// TIA Portal V20 export
VAR_GLOBAL   // PLC tag table "TROLLEY"
   mhUpperLimitSwitchBypassKeyCh1 AT %I300.0 : Bool;   // MH Upper limit Cam switch bypass key switch Channel 1
   mhUpperLimitSwitchBypassKeyCh2 AT %I300.4 : Bool;   // MH Upper limit Cam switch bypass key switch Channel 2
   mhUpperLimitSwitchBypassKeyCh1VS AT %I301.0 : Bool;   // MH Upper limit Cam switch bypass key switch Channel 1 Supply
   mhUpperLimitSwitchBypassKeyCh2VS AT %I301.4 : Bool;   // MH Upper limit Cam switch bypass key switch Channel 2 Supply
   mhLimitSwitchEmStopCh1 AT %I306.0 : Bool;   // MH Emergency stop limit switch Channel 1
   mh1LimitSwitchFRUEmStop AT %I306.1 : Bool;   // MH1 cam switch Raise emergency stop
   machineRoomDoorControlCh1 AT %I306.2 : Bool;   // Machine room door control switch Channel 1
   mh2LimitSwitchFRUEmStop AT %I306.3 : Bool;   // MH2 cam switch Raise emergency stop
   mhLimitSwitchEmStopCh2 AT %I306.4 : Bool;   // MH Emergency stop limit switch Channel 2
   mh1LimitSwitchBLDEmStop AT %I306.5 : Bool;   // MH1 cam switch Lower emergency stop
   machineRoomDoorControlCh2 AT %I306.6 : Bool;   // Machine room door control switch Channel 2
   mh2LimitSwitchBLDEmStop AT %I306.7 : Bool;   // MH2 cam switch Lower emergency stop
   machineRoomDoorControlCh1VS AT %I307.2 : Bool;   // Machine room door control switch Channel 1 supply
   mhLimitSwitchEmStopCh2VS AT %I307.4 : Bool;   // MH Emergency stop limit switch Channel 2 supply
   machineRoomDoorControlCh2VS AT %I307.6 : Bool;   // Machine room door control switch Channel 2 supply
   slewLimitSwitchBLDStopCh1 AT %I312.2 : Bool;   // Slewing limit switch Stop left Channel 1
   slewLimitSwitchFRUStopCh1 AT %I312.3 : Bool;   // Slewing limit switch Stop right Channel 1
   slewLimitSwitchBLDStopCh2 AT %I312.6 : Bool;   // Slewing limit switch Stop left Channel 2
   slewLimitSwitchFRUStopCh2 AT %I312.7 : Bool;   // Slewing limit switch Stop right Channel 2
   slewLimitSwitchBLDStopVS AT %I313.2 : Bool;   // Slewing limit switch Stop left Sensor supply
   slewLimitSwitchFRUStopVS AT %I313.3 : Bool;   // Slewing limit switch Stop right Sensor supply
   trolleyEntranceGateSouthControlCh1 AT %I318.2 : Bool;   // Trolley entrance gate south side control Channel 1
   trolleyEntranceGateNorthControlCh1 AT %I318.3 : Bool;   // Trolley entrance gate north side control Channel 1
   trolleyEntranceGateSouthControlCh2 AT %I318.6 : Bool;   // Trolley entrance gate south side control Channel 2
   trolleyEntranceGateNorthControlCh2 AT %I318.7 : Bool;   // Trolley entrance gate north side control Channel 2
   trolleyEntranceGateSouthControlCh1VS AT %I319.2 : Bool;   // Trolley entrance gate south side control Channel 1 supply
   trolleyEntranceGateNorthControlCh1VS AT %I319.3 : Bool;   // Trolley entrance gate north side control Channel 1 supply
   trolleyEntranceGateSouthControlCh2VS AT %I319.6 : Bool;   // Trolley entrance gate south side control Channel 2 supply
   trolleyEntranceGateNorthControlCh2VS AT %I319.7 : Bool;   // Trolley entrance gate north side control Channel 2 supply
   btnEmStopRopeChangeBoxCh1 AT %I324.2 : Bool;   // Rope change box Emergency stop Channel 1
   ropeChangeBoxHoldToRunBtnCh1 AT %I324.3 : Bool;   // Rope change box Hold-to-run button Channel 1
   btnEmStopRopeChangeBoxCh2 AT %I324.6 : Bool;   // Rope change box Emergency stop Channel 2
   ropeChangeBoxHoldToRunBtnCh2 AT %I324.7 : Bool;   // Rope change box Hold-to-run button Channel 2
   btnEmStopRopeChangeBoxCh1VS AT %I325.2 : Bool;   // Rope change box Emergency stop Channel 1 Supply
   ropeChangeBoxHoldToRunBtnCh1VS AT %I325.3 : Bool;   // Rope change box Hold-to-run button Channel 1 Supply
   btnEmStopRopeChangeBoxCh2VS AT %I325.6 : Bool;   // Rope change box Emergency stop Channel 2 Supply
   ropeChangeBoxHoldToRunBtnCh2VS AT %I325.7 : Bool;   // Rope change box Hold-to-run button Channel 2 Supply
   cabinPlatformGateTrolleySideControlCh1 AT %I330.1 : Bool;   // Cabin platform gate (trolley side) control Channel 1
   btnEmStopSpreader AT %I330.2 : Bool;   // Spreader Emergency stop
   cabinEntranceInterlockMagnetPosCh1 AT %I330.3 : Bool;   // Cabin entrance interlock magnet position Channel 1
   cabinPlatformGateTrolleySideControlCh2 AT %I330.5 : Bool;   // Cabin platform gate (trolley side) control Channel 2
   limitSwitchSpreaderAntiTwoBlock AT %I330.6 : Bool;   // Spreader anti-two block emergency switch
   cabinEntranceInterlockMagnetPosCh2 AT %I330.7 : Bool;   // Cabin entrance interlock magnet position Channel 2
   cabinPlatformGateTrolleySideControlCh1VS AT %I331.1 : Bool;   // Cabin platform gate (trolley side) control Channel 1 supply
   btnEmStopSpreaderVS AT %I331.2 : Bool;   // Spreader Emergency stop Channel supply
   cabinPlatformGateTrolleySideControlCh2VS AT %I331.5 : Bool;   // Cabin platform gate (trolley side) control Channel 2 supply
   limitSwitchSpreaderAntiTwoBlockVS AT %I331.6 : Bool;   // Spreader anti-two block emergency switch Channel supply
   spare AT %I360.1 : Bool;   // Spare
   cbIllumSocketsTrolley AT %I360.2 : Bool;   // Illumination/sockets trolley CB Feedback
   cb230VCircuitsTrolley AT %I360.3 : Bool;   // 230V circuits trolley CB Feedback
   cbCabin400VLoads AT %I360.4 : Bool;   // Cabin 400V loads CB Feedback
   cbCabin230VLoads AT %I360.5 : Bool;   // Cabin 230V loads CB Feedback
   cbIllumTrolleyRCB AT %I360.6 : Bool;   // Illumination Trolley RCB Feedback
   cbTrolleySockets400VRCBO AT %I360.7 : Bool;   // Trolley Sockets 400V RCBO Feedback
   cbTrolleySockets230VRCBO AT %I361.0 : Bool;   // Trolley Sockets 230V RCBO Feedback
   cbIllumTrolleyMachineRoom AT %I361.1 : Bool;   // Illumination Trolley machine room CB Feedback
   cbIllumTrolleyWalkways AT %I361.2 : Bool;   // Illumination Trolley walkways CB Feedback
   cbIllumTrolleyFloodLight AT %I361.3 : Bool;   // Illumination Trolley flood light CB Feedback
   cbUpsOutput AT %I361.4 : Bool;   // UPS output CB Feedback
   illumTrolleyFloodLightMCStarted AT %I361.5 : Bool;   // Illumination Trolley flood light contactor Feedback
   upsTrolleyFloodAlarm AT %I361.6 : Bool;   // Trolley flood UPS Alarm
   upsTrolleyFloodBatteryMode AT %I361.7 : Bool;   // Trolley flood UPS Battery mode
   cb24trolleyPS AT %I362.0 : Bool;   // 24VDC Trolley PS CB Feedback
   trolleyPS24OK AT %I362.1 : Bool;   // 24VDC Trolley PS OK
   ups24trolleyBatteryMode AT %I362.2 : Bool;   // 24VDC Trolley UPS Battery mode
   ups24trolleyOK AT %I362.3 : Bool;   // 24VDC Trolley UPS 24VDC OK
   ups24trolleyAlarm AT %I362.4 : Bool;   // 24VDC Trolley UPS Alarm
   ups24trolleyReadyToBuffer AT %I362.5 : Bool;   // 24VDC Trolley UPS Ready to buffer
   ups24trolleyBatGt85 AT %I362.6 : Bool;   // 24VDC Trolley UPS BAT.>85%
   "cbPnSwitchSupply(1)" AT %I362.7 : Bool;   // PN switch supply CB Feedback
   cb24Spare AT %I363.0 : Bool;   // 24 VDC CB Spare Feedback
   "cbAccessCircuits(1)" AT %I363.1 : Bool;   // Access circuits CB Feedback
   cbMotorProtectionRelays AT %I363.2 : Bool;   // Motor protection relays, optic transmitters CB Feedback
   cbMhSensorsSupply AT %I363.3 : Bool;   // MH sensors supply CB Feedback
   "cbCtSensorsSupply(1)" AT %I363.4 : Bool;   // CT sensors supply CB Feedback
   cbSlewSensorsSupply AT %I363.5 : Bool;   // Slewing sensors supply CB Feedback
   cbWindTransmitterSupply AT %I363.6 : Bool;   // Wind transmitter supply CB Feedback
   cbTelephoneSystemTrolley AT %I363.7 : Bool;   // Telephone system supply trolley CB Feedback
   cbLehnertSystem AT %I364.0 : Bool;   // LEHNERT system CB Feedback
   cbLaseIPCSupply AT %I364.1 : Bool;   // LASE IPC supply CB Feedback
   cb230Spare AT %I364.2 : Bool;   // 230V spare CB Feedback
   "cb230Spare(1)" AT %I364.3 : Bool;   // 230V spare CB Feedback
   "cb24Spare(1)" AT %I364.4 : Bool;   // 24VDC spare CB Feedback
   "cb24Spare(2)" AT %I364.5 : Bool;   // 24VDC spare CB Feedback
   cbSiren AT %I364.6 : Bool;   // Siren CB Feedback
   trolleyCoolingFanMCStarted AT %I365.4 : Bool;   // Trolley machine room cooling fan contactor Feedback
   trolleyHeaterMCStarted AT %I365.5 : Bool;   // Trolley machine room heater contactor Feedback
   cbCabinCtrlCircuits24VS AT %I365.6 : Bool;   // Cabin control circuits 24VDC Supply CB Feedback
   cbMh1Brake AT %I366.0 : Bool;   // MH1 Brake CB Feedback
   cbMh1ForcedCoolingFan AT %I366.1 : Bool;   // MH1 Forced cooling fan CB Feedback
   cbMh1AntiCondHeating AT %I366.2 : Bool;   // MH1 Anti- condensation heating CB Feedback
   mh1CoolingFanMCStarted AT %I366.3 : Bool;   // MH1 Forced cooling fan contactor Feedback
   "cbMh1AntiCondHeating(1)" AT %I366.4 : Bool;   // MH1 Anti-condensation heating CB Feedback
   mh1BrakeMC1Started AT %I366.5 : Bool;   // MH1 brake contactor 1 feedback
   mh1BrakeMC2Started AT %I366.6 : Bool;   // MH1 brake contactor 2 feedback
   mh1BrakeOpen AT %I366.7 : Bool;   // MH1 Brake Open
   mh1BrakeWear AT %I367.0 : Bool;   // MH1 Brake Wear
   mh1LimitSwitchFRUStop AT %I367.1 : Bool;   // MH1 cam switch Raise end stop
   mh1LimitSwitchFRUSlowDown AT %I367.2 : Bool;   // MH1 cam switch Raise speed reduction
   mh1LimitSwitchBLDStop AT %I367.3 : Bool;   // MH1 cam switch Lower end stop
   mh1LimitSwitchBLDSlowDown AT %I367.4 : Bool;   // MH1 cam switch Lower speed reduction
   ropeDescendRelay1 AT %I367.6 : Bool;   // Rope descend relay 1
   ropeDescendRelay2 AT %I367.7 : Bool;   // Rope descend relay 2
   cbMh2Brake AT %I368.0 : Bool;   // MH2 Brake CB Feedback
   cbMh2ForcedCoolingFan AT %I368.1 : Bool;   // MH2 Forced cooling fan CB Feedback
   cbMh2AntiCondHeating AT %I368.2 : Bool;   // MH2 Anti- condensation heating CB Feedback
   mh2CoolingFanMCStarted AT %I368.3 : Bool;   // MH2 Forced cooling fan contactor Feedback
   "cbMh2AntiCondHeating(1)" AT %I368.4 : Bool;   // MH2 Anti-condensation heating CB Feedback
   mh2BrakeMC1Started AT %I368.5 : Bool;   // MH2 brake contactor 1 feedback
   mh2BrakeMC2Started AT %I368.6 : Bool;   // MH2 brake contactor 2 feedback
   mh2BrakeOpen AT %I368.7 : Bool;   // MH2 Brake Open
   mh2BrakeWear AT %I369.0 : Bool;   // MH2 Brake Wear
   mh2LimitSwitchFRUStop AT %I369.1 : Bool;   // MH2 cam switch Raise end stop
   mh2LimitSwitchFRUSlowDown AT %I369.2 : Bool;   // MH2 cam switch Raise speed reduction
   mh2LimitSwitchBLDStop AT %I369.3 : Bool;   // MH2 cam switch Lower end stop
   mh2LimitSwitchBLDSlowDown AT %I369.4 : Bool;   // MH2 cam switch Lower speed reduction
   "spare(1)" AT %I369.7 : Bool;   // Spare
   cbCtBrakes AT %I370.0 : Bool;   // CT Brakes CB Feedback
   cbCtAntiCondHeating AT %I370.1 : Bool;   // CT Anti-condensation heating CB Feedback
   ctAntiCondHeatingMCStarted AT %I370.2 : Bool;   // CT Anti-condensation heating contactor Feedback
   ct1Motor1TempCtrl AT %I370.5 : Bool;   // CT1 motor 1 temperature control
   ct1Motor2TempCtrl AT %I370.6 : Bool;   // CT1 motor 2 temperature control
   ct2Motor1TempCtrl AT %I370.7 : Bool;   // CT2 motor 1 temperature control
   ct2Motor2TempCtrl AT %I371.0 : Bool;   // CT2 motor 2 temperature control
   "spare(2)" AT %I371.1 : Bool;   // Spare
   "spare(3)" AT %I371.2 : Bool;   // Spare
   "spare(4)" AT %I371.3 : Bool;   // Spare
   "spare(5)" AT %I371.4 : Bool;   // Spare
   "spare(6)" AT %I371.5 : Bool;   // Spare
   "spare(7)" AT %I371.6 : Bool;   // Spare
   "spare(8)" AT %I371.7 : Bool;   // Spare
   cbSlewBrakes AT %I372.0 : Bool;   // Slewing brakes CB Feedback
   cbSlewAntiCondHeating AT %I372.1 : Bool;   // Slewing anti-condensation heating CB Feedback
   slewAntiCondHeatingMCStarted AT %I372.2 : Bool;   // Slewing anti-condensation heating contactor Feedback
   slewBrakesControlMC1Started AT %I372.3 : Bool;   // Slewing brakes control Contactor 1 feedback
   slewBrakesControlMC2Started AT %I372.4 : Bool;   // Slewing brakes control Contactor 2 feedback
   slewMotor1TempCtrl AT %I372.5 : Bool;   // Slewing motor 1 temperature control
   slewMotor2TempCtrl AT %I372.6 : Bool;   // Slewing motor 2 temperature control
   cbKstBoxSupply AT %I373.0 : Bool;   // KST box supply CB Feedback
   loadMomentGt115 AT %I373.1 : Bool;   // Load moment>115%
   loadMomentGt105 AT %I373.2 : Bool;   // Load moment>105%
   loadMomentGt95 AT %I373.3 : Bool;   // Load moment>95%
   loadGt11t AT %I373.4 : Bool;   // Load>11t
   maxUnitLoad AT %I373.5 : Bool;   // Max. unit load
   excenterAbMinusCd AT %I373.6 : Bool;   // Excenter (A+B)-(C+D)
   ropeLoop AT %I373.7 : Bool;   // Rope loop
   cbSpreaderHydraulicPump1 AT %I374.0 : Bool;   // Spreader Hydraulic pump 1 CB Feedback
   cbSpreaderHydraulicPump2 AT %I374.1 : Bool;   // Spreader Hydraulic pump 2 CB Feedback
   cbSpreaderHeating230Vac AT %I374.2 : Bool;   // Spreader Heating power supply 230VAC CB Feedback
   cbSpreaderControl230Vac AT %I374.3 : Bool;   // Spreader Control voltage 230VAC CB Feedback
   cb24SpreaderSupply AT %I374.4 : Bool;   // Spreader 24VDC power supply CB Feedback
   cbSpreaderEmStopRelays AT %I374.5 : Bool;   // Spreader emergency stop relays CB Feedback
   cbLaseCabinet230V AT %I374.6 : Bool;   // LASE cabinet 230V supply CB Feedback
   "cabinEntranceInterlockMagnetPosNO(1)" AT %I375.0 : Bool;   // Cabin entrance interlock magnet position signaling contact (NO)
   lockOpenBtnCabinSide AT %I375.1 : Bool;   // Lock opening button cabin side
   cabinEntranceDoorInterlockMCStarted AT %I375.2 : Bool;   // Cabin entrance door interlock contactor Feedback
   machineRoomDoorControlFb AT %I375.3 : Bool;   // Machine room door control switch Feedback
   cabinPlatformGateTrolleySideControlFb AT %I375.4 : Bool;   // Cabin platform gate (trolley side) control Feedback
   trolleyEntranceGateSouthControlFb AT %I375.5 : Bool;   // Trolley entrance gate south side control Feedback
   trolleyEntranceGateNorthControlFb AT %I375.6 : Bool;   // Trolley entrance gate north side control Feedback
   trolleyExitGateStairsControl AT %I375.7 : Bool;   // Trolley exit to the stairs gate control
   ropeChangeBoxStart AT %I376.0 : Bool;   // Rope change box Start rope change
   ropeChangeBoxSiren AT %I376.1 : Bool;   // Rope change box Siren control
   ropeChangeBoxMhFRU AT %I376.2 : Bool;   // Rope change box MH up
   ropeChangeBoxMhBLD AT %I376.3 : Bool;   // Rope change box MH down
   ropeChangeBoxCtFRU AT %I376.4 : Bool;   // Rope change box CT forward
   ropeChangeBoxCtBLD AT %I376.5 : Bool;   // Rope change box CT backward
   ropeChangeBoxSlewBLD AT %I376.6 : Bool;   // Rope change box Slewing left rotation
   ropeChangeBoxSlewFRU AT %I376.7 : Bool;   // Rope change box Slewing right rotation
   ropeChangeBoxCtParking AT %I377.0 : Bool;   // Rope change box Cross travel to parking position
   cbLubricationStation230V AT %I377.1 : Bool;   // Lubrication station 230V supply CB Feedback
   lubricationEnable AT %I377.2 : Bool;   // Lubrication station enable
   "spare(9)" AT %I377.3 : Bool;   // Spare
   windAlarmWarning AT %I377.6 : Bool;   // Wind Alarm Unit Warning
   "windAlarmWarning(1)" AT %I377.7 : Bool;   // Wind Alarm Unit Warning
   cbJackScrewMotorNorth AT %I378.0 : Bool;   // Jack-screw motor North side CB Feedback
   jackScrewNorthMCFRUStarted AT %I378.1 : Bool;   // Jack-screw motor North side contactor up Feedback
   jackScrewNorthMCBLDStarted AT %I378.2 : Bool;   // Jack-screw motor North side contactor down Feedback
   cbJackScrewMotorSouth AT %I378.3 : Bool;   // Jack-screw motor South side CB Feedback
   jackScrewSouthMCFRUStarted AT %I378.4 : Bool;   // Jack-screw motor South side contactor up Feedback
   jackScrewSouthMCBLDStarted AT %I378.5 : Bool;   // Jack-screw motor South side contactor down Feedback
   jackScrewNorthMotorTempCtrl AT %I378.6 : Bool;   // Jack-screw north side motor temperature control
   jackScrewSouthMotorTempCtrl AT %I378.7 : Bool;   // Jack-screw south side motor temperature control
   jackScrewNorthUpperPos AT %I379.0 : Bool;   // Jack-screw North side Upper position
   jackScrewNorthLowerPos AT %I379.1 : Bool;   // Jack-screw North side Lower position
   jackScrewSouthUpperPos AT %I379.2 : Bool;   // Jack-screw South side Upper position
   jackScrewSouthLowerPos AT %I379.3 : Bool;   // Jack-screw South side Lower position
   slewBrakeMC1Start AT %Q341.2 : Bool;   // Slewing brakes control Contactor 1
   slewBrakeMC2Start AT %Q341.3 : Bool;   // Slewing brakes control Contactor 2
   spreaderEmStopRelay AT %Q346.0 : Bool;   // Spreader emergency stop relay
   cabinEntranceDoorInterlockMCStart AT %Q346.1 : Bool;   // Cabin entrance door interlock control
   sirenStart AT %Q360.0 : Bool;   // Siren control relay
   mh1CoolingFanMCStart AT %Q360.1 : Bool;   // MH1 cooling fan Contactor
   mh1AntiCondMCStart AT %Q360.2 : Bool;   // MH1 anti-condensation heating Contactor
   mh2CoolingFanMCStart AT %Q360.3 : Bool;   // MH2 cooling fan Contactor
   mh2AntiCondMCStart AT %Q360.4 : Bool;   // MH2 anti-condensation heating Contactor
   ctAntiCondMCStart AT %Q360.5 : Bool;   // CT Anti-condensation heating control Contactor
   slewAntiCondMCStart AT %Q360.6 : Bool;   // Slewing anti-condensation heating control Contactor
   illumTrolleyWalkwaysMCStart AT %Q361.0 : Bool;   // Illumination Trolley walkways ON/OFF (impulse control)
   illumTrolleyFloodLightMCStart AT %Q361.3 : Bool;   // Illumination Trolley flood light ON/OFF (impulse control)
   lubricationStart AT %Q361.6 : Bool;   // Lubrication station control
   lubricationAddStart AT %Q361.7 : Bool;   // Lubrication station Additional lubrication
   jackScrewNorthMCFRUStart AT %Q362.0 : Bool;   // Jack-screw motor North side contactor up
   jackScrewNorthMCBLDStart AT %Q362.1 : Bool;   // Jack-screw motor North side contactor down
   jackScrewSouthMCFRUStart AT %Q362.2 : Bool;   // Jack-screw motor South side contactor up
   jackScrewSouthMCBLDStart AT %Q362.3 : Bool;   // Jack-screw motor South side contactor down
   iMh1MotorTemp1 AT %IW380 : Int;   // MH1 motor temperature sensor 1
   iMh1MotorTemp2 AT %IW382 : Int;   // MH1 motor temperature sensor 2
   iMh2MotorTemp1 AT %IW384 : Int;   // MH2 motor temperature sensor 1
   iMh2MotorTemp2 AT %IW386 : Int;   // MH2 motor temperature sensor 2
   iMainLoadPin1Out AT %QW364 : Int;   // Main load pin 1
   iMainLoadPin2Out AT %QW366 : Int;   // Main load pin 2
   iMainLoadPin3Out AT %QW368 : Int;   // Main load pin 3
   iMainLoadPin4Out AT %QW370 : Int;   // Main load pin 4
   iRedundantLoadPin1Out AT %QW372 : Int;   // Redundant load pin 1
   iRedundantLoadPin2Out AT %QW374 : Int;   // Redundant load pin 2
   iRedundantLoadPin3Out AT %QW376 : Int;   // Redundant load pin 3
   iRedundantLoadPin4Out AT %QW378 : Int;   // Redundant load pin 4
   btnEmStopTrolleyNorthCh2VS AT %I325.4 : Bool;   // Trolley Emergency stop North side Channel 2 Supply
   btnEmStopTrolleyNorthCh1VS AT %I325.0 : Bool;   // Trolley Emergency stop North side Channel 1 Supply
   spare1Ch1 AT %I318.0 : Bool;   // Spare Channel 1
   btnEmStopTrolleyCabinetCh1VS AT %I301.1 : Bool;   // Trolley cabinet Emergency stop Channel 1
   btnEmStopTrolleyNorthCh2 AT %I324.4 : Bool;   // Trolley Emergency stop North side Channel 2
   btnEmStopTrolleyCabinetCh2 AT %I300.5 : Bool;   // Trolley cabinet Emergency stop Channel 2
   spare1Ch2VS AT %I319.4 : Bool;   // Spare Channel 2 Supply
   spare1Ch1VS AT %I319.0 : Bool;   // Spare Channel 1 Supply
   btnEmStopTrolleyCabinetCh2VS AT %I301.5 : Bool;   // Trolley cabinet Emergency stop Channel 2
   spare1Ch2 AT %I318.4 : Bool;   // Spare Channel 2
   spare2Ch1 AT %I318.1 : Bool;   // Spare Channel 1
   btnEmStopTrolleyNorthCh1 AT %I324.0 : Bool;   // Trolley Emergency stop North side Channel 1
   btnEmStopTrolleySouthCh2 AT %I324.5 : Bool;   // Trolley Emergency stop South side Channel 2
   mhLimitSwitchEmStopCh1VS AT %I307.0 : Bool;   // MH Emergency stop limit switch Channel 1
   spare2Ch2 AT %I318.5 : Bool;   // Spare Channel 2
   spare2Ch2VS AT %I319.5 : Bool;   // Spare Channel 2 Supply
   btnEmStopTrolleyCabinetCh1 AT %I300.1 : Bool;   // Trolley cabinet Emergency stop Channel 1
   btnEmStopTrolleySouthCh1VS AT %I325.1 : Bool;   // Trolley Emergency stop South side Channel 1 Supply
   btnEmStopTrolleySouthCh2VS AT %I325.5 : Bool;   // Trolley Emergency stop South side Channel 2 Supply
   spare2Ch1VS AT %I319.1 : Bool;   // Spare Channel 1 Supply
   btnEmStopTrolleySouthCh1 AT %I324.1 : Bool;   // Trolley Emergency stop South side Channel 1
   mh2BrakeMC1Start AT %Q336.2 : Bool;   // MH2 brake Contactor 1
   ctBrakeMC2Start AT %Q341.1 : Bool;   // CT brakes control Contactor 2
   mh1BrakeMC2Start AT %Q336.1 : Bool;   // MH1 brake Contactor 2
   mh1BrakeMC1Start AT %Q336.0 : Bool;   // MH1 brake Contactor 1
   ctBrakeMC1Start AT %Q341.0 : Bool;   // CT brakes control Contactor 1
   ctBrakesMC1Started AT %I370.3 : Bool;   // CT brakes control Contactor 1 feedback
   mh2BrakeMC2Start AT %Q336.3 : Bool;   // MH2 brake Contactor 2
   ctBrakesMC2Started AT %I370.4 : Bool;   // CT brakes control Contactor 2 feedback
   illumTrolleyMachineRoomMCStart AT %Q360.7 : Bool;   // Illumination Trolley machine room ON/OFF (impulse control)
   "cbTrolleyMachineRoomHeater(1)" AT %I365.2 : Bool;   // Trolley machine room heater CB Feedback
   "cbTrolleyMachineRoom230VCtrl(1)" AT %I365.3 : Bool;   // Trolley machine room 230V control circuit CB Feedback
   "cbTrolley400VLoadsTrolleyCabinet(1)" AT %I360.0 : Bool;   // Trolley 400V loads CB (Trolley cabinet) Feedback
   "cbTrolleyMachineRoomCoolingFan(1)" AT %I365.1 : Bool;   // Trolley machine room cooling fan CB Feedback
END_VAR
